% RSLogix 500 project THREE-PHASE MOTOR CONTROL_BAK003.RSS, saved by version 10.00.00.00 %
PROJECT "MRLEIGH"    % processor: Bul.1763 MicroLogix 1100 Series B %

PROGRAM FILES
  LAD 2 "INV"  4 rungs  % Invert Signals Wired Failsafe %
  LAD 3 "SIM"  2 rungs  % Simulation Program %
  LAD 4 "MAN"  5 rungs  % Main Program %

DATA FILES
  O0 OUTPUT  4 elements
  I1 INPUT  6 elements
  S2 STATUS  66 elements
  B3 BINARY  1 elements
  T4 TIMER  1 elements
  C5 COUNTER  1 elements
  R6 CONTROL  1 elements
  N7 INTEGER  1 elements
  F8 FLOAT  1 elements

LADDER 2 "INV"    % Invert Signals Wired Failsafe %
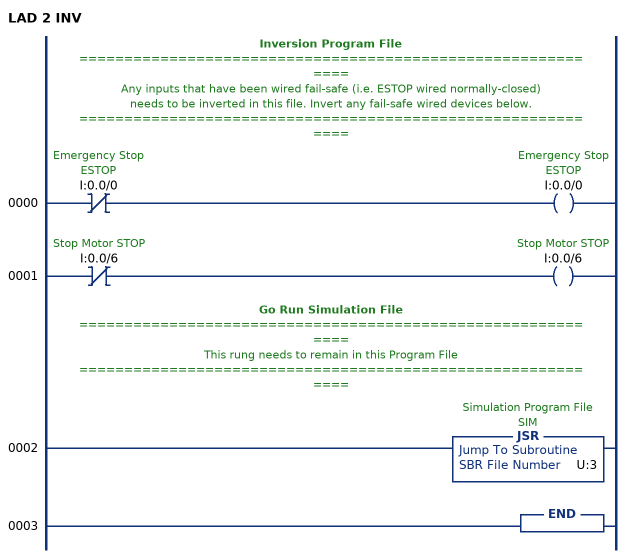
% Rung: 0 %
% TITLE: Inversion Program File %
% ============================================================
% 
%   Any inputs that have been wired fail-safe (i.e. ESTOP wired normally-closed)
%   needs to be inverted in this file. Invert any fail-safe wired devices below.
% 
% ============================================================ %
SOR XIO I:0.0/0 OTE I:0.0/0 EOR
%   I:0.0/0  ESTOP  "Emergency Stop" %
% Rung: 1 %
SOR XIO I:0.0/6 OTE I:0.0/6 EOR
%   I:0.0/6  STOP  "Stop Motor" %
% Rung: 2 %
% TITLE: Go Run Simulation File %
% ============================================================
% 
%   This rung needs to remain in this Program File
% 
% ============================================================ %
SOR JSR U:3 EOR
%   U:3  SIM  "Simulation Program File" %
% Rung: 3 %
SOR END EOR

LADDER 3 "SIM"    % Simulation Program %
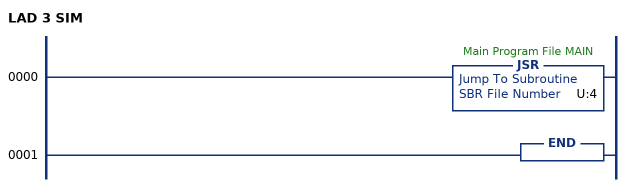
% Rung: 0 %
SOR JSR U:4 EOR
%   U:4  MAIN  "Main Program File" %
% Rung: 1 %
SOR END EOR

LADDER 4 "MAN"    % Main Program %
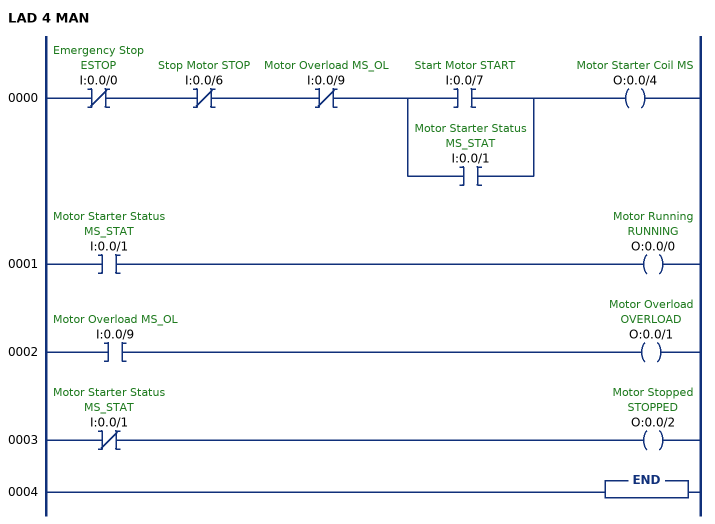
% Rung: 0 %
SOR XIO I:0.0/0 XIO I:0.0/6 XIO I:0.0/9 BST XIC I:0.0/7 NXB XIC I:0.0/1 BND OTE O:0.0/4 EOR
%   I:0.0/0  ESTOP  "Emergency Stop" %
%   I:0.0/6  STOP  "Stop Motor" %
%   I:0.0/9  MS_OL  "Motor Overload" %
%   I:0.0/7  START  "Start Motor" %
%   I:0.0/1  MS_STAT  "Motor Starter Status" %
%   O:0.0/4  MS  "Motor Starter Coil" %
% Rung: 1 %
SOR XIC I:0.0/1 OTE O:0.0/0 EOR
%   I:0.0/1  MS_STAT  "Motor Starter Status" %
%   O:0.0/0  RUNNING  "Motor Running" %
% Rung: 2 %
SOR XIC I:0.0/9 OTE O:0.0/1 EOR
%   I:0.0/9  MS_OL  "Motor Overload" %
%   O:0.0/1  OVERLOAD  "Motor Overload" %
% Rung: 3 %
SOR XIO I:0.0/1 OTE O:0.0/2 EOR
%   I:0.0/1  MS_STAT  "Motor Starter Status" %
%   O:0.0/2  STOPPED  "Motor Stopped" %
% Rung: 4 %
SOR END EOR

OTHER DOCUMENTED ADDRESSES
  PFILE:3  "Simulation"
